// TIA Portal V20 export
DATA_BLOCK "LPFE_PerformanceMeasurement"   // DB277
TITLE = PerformanceTest
{ DB_Accessible_From_OPC_UA := 'FALSE' }
// Stores the measured round trip times from messages that are requested and responded by the request handler
// stored: Access Published, DBAccessibleFromOPCUA false, MemoryReserve 100, Namespace PFE
   VAR
      performanceMeasurement { ExternalAccessible := 'False'; ExternalVisible := 'False'; ExternalWritable := 'False'} : Array[0.._.LE_NUMBER_OF_INTERFACE_BUFFERS] of "LPFE_typeRequestMeasureBuffer";   // Each handler has its own performance measurements
   END_VAR
BEGIN
END_DATA_BLOCK
